{attribute 'no-analysis'}
{attribute 'qualified_only'} 
VAR_GLOBAL
	{attribute 'hide'} 
	aBuffer:				ARRAY[0..99] OF FB_Message;
	{attribute 'hide'} 
    nBuffer:				UINT := 0;
	{attribute 'hide'} 
	nTimestamp:				Tc2_Utilities.T_FILETIME64;	
	{attribute 'hide'} 
	nFunction:				Tc2_Utilities.T_FILETIME64;		
END_VAR

(* stored: Version 1.1.0.1
   GVL GVL: Id {8c417638-2928-4f7d-b718-658b035f50d1} *)
